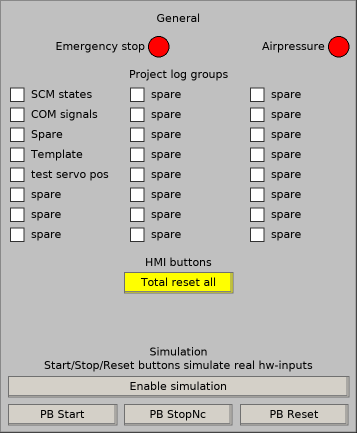
VISUALIZATION Vis_General  // 357x433
VAR_IN_OUT
	IO_General: utl_General;
END_VAR
    Rectangle (0,0 357x433)
    Rectangle (8,8 341x21), "General"
    Button (8,376 341x21), "Enable simulation"
        toggle Glbl.SimEnable
    Button (124,272 109x21), "Total reset all", pressed state: IO_General.PbSf_TotalResetAll.P_BypassStateTrue
        tap IO_General.PbSf_TotalResetAll.P_BypassStateTrue
    Checkbox (8,84 21x21), variable: BknLog.ActiveGroups.8
    Checkbox (8,104 21x21), variable: BknLog.ActiveGroups.9
    Checkbox (8,124 21x21), variable: BknLog.ActiveGroups.10
    Checkbox (8,164 21x21), variable: BknLog.ActiveGroups.12
    Checkbox (8,184 21x21), variable: BknLog.ActiveGroups.13
    Checkbox (8,204 21x21), variable: BknLog.ActiveGroups.14
    Checkbox (8,144 21x21), variable: BknLog.ActiveGroups.11
    Checkbox (8,224 21x21), variable: BknLog.ActiveGroups.15
    Label (28,84 81x21), "SCM states"
    Label (8,64 341x21), "Project log groups"
    Label (28,104 81x21), "COM signals"
    Label (28,124 81x21), "Spare"
    Label (28,144 81x21), "Template"
    Label (28,164 81x21), "test servo pos"
    Label (28,184 81x21), "spare"
    Label (28,204 81x21), "spare"
    Label (28,224 81x21), "spare"
    Checkbox (128,204 21x21), variable: BknLog.ActiveGroups.22
    Checkbox (128,224 21x21), variable: BknLog.ActiveGroups.23
    Checkbox (248,84 21x21), variable: BknLog.ActiveGroups.24
    Checkbox (128,184 21x21), variable: BknLog.ActiveGroups.21
    Checkbox (248,104 21x21), variable: BknLog.ActiveGroups.25
    Label (148,184 81x21), "spare"
    Label (148,204 81x21), "spare"
    Label (148,224 81x21), "spare"
    Label (268,84 81x21), "spare"
    Label (268,104 81x21), "spare"
    Checkbox (128,124 21x21), variable: BknLog.ActiveGroups.18
    Checkbox (128,144 21x21), variable: BknLog.ActiveGroups.19
    Checkbox (128,164 21x21), variable: BknLog.ActiveGroups.20
    Label (148,124 81x21), "spare"
    Label (148,144 81x21), "spare"
    Label (148,164 81x21), "spare"
    Checkbox (128,84 21x21), variable: BknLog.ActiveGroups.16
    Checkbox (128,104 21x21), variable: BknLog.ActiveGroups.17
    Label (148,84 81x21), "spare"
    Label (148,104 81x21), "spare"
    Checkbox (248,124 21x21), variable: BknLog.ActiveGroups.26
    Checkbox (248,144 21x21), variable: BknLog.ActiveGroups.27
    Label (268,124 81x21), "spare"
    Label (268,144 81x21), "spare"
    Checkbox (248,164 21x21), variable: BknLog.ActiveGroups.28
    Checkbox (248,184 21x21), variable: BknLog.ActiveGroups.29
    Label (268,164 81x21), "spare"
    Label (268,184 81x21), "spare"
    Checkbox (248,204 21x21), variable: BknLog.ActiveGroups.30
    Checkbox (248,224 21x21), variable: BknLog.ActiveGroups.31
    Label (268,204 81x21), "spare"
    Label (268,224 81x21), "spare"
    Rectangle (8,340 341x37), "Simulation Start/Stop/Reset buttons simulate real hw-inputs"
    Button (8,404 109x21), "PB Start"
        tap MAIN.General.I_Pb_StartAll.I_K_SimulateOn
    Button (124,404 108x21), "PB StopNc"
        toggle MAIN.General.I_PbNc_StopAll.I_K_SimulateOn
    Button (240,404 108x21), "PB Reset"
        tap MAIN.General.I_Pb_ResetAll.I_K_SimulateOn
    Label (8,252 341x21), "HMI buttons"
    Ellipse (148,36 21x21), colour toggle: IO_General.Q_SN_ES_Zone1_OK
    Label (0,36 148x21), "Emergency stop"
    Label (180,36 148x21), "Airpressure"
    Ellipse (328,36 21x21), colour toggle: MAIN.General.I_PS_AirpressureOk.HMI.STS.State
END_VISUALIZATION

(* stored: Version 1.1.0.1
   Visu Vis_General: Id {2100ec78-39f2-419c-8e0b-cf8dddf3b2a2} *)
